{attribute 'linkalways'}
{attribute 'no_explicit_call' := 'This FB is a CLASS and must be accessed using methods or properties'}
{attribute 'enable_dynamic_creation'}
FUNCTION_BLOCK Node_F_VN_LocateCircularArcExp2 EXTENDS VisionNode
VAR
    ipSrcImage : _ITcVnImage;
    stCircularArc : _TcVnCircularArc;
    aCenter : _TcVnPoint2_REAL;
    fSearchRadius : _REAL(0.0);
    fArcDirectionRad : _LREAL(0.0);
    eEdgeDirection : _ETcVnEdgeDirection(ETcVnEdgeDirection.TCVN_ED_DARK_TO_LIGHT);
    fMinStrength : _REAL(0.0);
    fAngleStepRad : _LREAL(0.1);
    nMaxThickness : _UDINT(10);
    bInvertSearchDirection : _BOOL(FALSE);
    nSubpixelsIterations : _UDINT(10);
    fApproxPrecision : _REAL(0.001);
    eAlgorithm : _ETcVnEdgeDetectionAlgorithm(ETcVnEdgeDetectionAlgorithm.TCVN_EDA_INTERPOLATION);
    ipContourPoints : _ITcVnContainer;
    fRangeCutoffFactor : _REAL(0.135);
    hrPrev : _HRESULT(S_OK);
    hresult : _HRESULT(S_OK);
END_VAR

METHOD PUBLIC Clone : I_Node
VAR
    pNode : POINTER TO Node_F_VN_LocateCircularArcExp2;
END_VAR
pNode := __NEW(Node_F_VN_LocateCircularArcExp2);
Clone := pNode^;
END_METHOD

METHOD FB_init : BOOL
VAR_INPUT
    bInitRetains : BOOL;
    bInCopyCode : BOOL;
END_VAR
AddInput('ipSrcImage', ipSrcImage);
AddOutput('stCircularArc', stCircularArc);
AddInput('aCenter', aCenter);
AddParameter('fSearchRadius', fSearchRadius);
AddParameter('fArcDirectionRad', fArcDirectionRad);
AddParameter('eEdgeDirection', eEdgeDirection);
AddParameter('fMinStrength', fMinStrength);
AddParameter('fAngleStepRad', fAngleStepRad);
AddParameter('nMaxThickness', nMaxThickness);
AddParameter('bInvertSearchDirection', bInvertSearchDirection);
AddParameter('nSubpixelsIterations', nSubpixelsIterations);
AddParameter('fApproxPrecision', fApproxPrecision);
AddParameter('eAlgorithm', eAlgorithm);
AddOutput('ipContourPoints', ipContourPoints);
AddParameter('fRangeCutoffFactor', fRangeCutoffFactor);
AddInput('hrPrev', hrPrev);
AddOutput('aCenter', aCenter);
AddOutput('hresult', hresult);
END_METHOD

METHOD PROTECTED OnExecute
hresult.Value := F_VN_LocateCircularArcExp2(
    ipSrcImage := ipSrcImage.Value,
    stCircularArc := stCircularArc.Value,
    aCenter := aCenter.Value,
    fSearchRadius := fSearchRadius.Value,
    fArcDirectionRad := fArcDirectionRad.Value,
    eEdgeDirection := eEdgeDirection.Value,
    fMinStrength := fMinStrength.Value,
    fAngleStepRad := fAngleStepRad.Value,
    nMaxThickness := nMaxThickness.Value,
    bInvertSearchDirection := bInvertSearchDirection.Value,
    nSubpixelsIterations := nSubpixelsIterations.Value,
    fApproxPrecision := fApproxPrecision.Value,
    eAlgorithm := eAlgorithm.Value,
    ipContourPoints := ipContourPoints.Value,
    fRangeCutoffFactor := fRangeCutoffFactor.Value,
    hrPrev := hrPrev.Value);
END_METHOD

METHOD PUBLIC PreExecutionCheck
VAR_INPUT
    Check : I_PreExecutionChecks;
END_VAR
VAR
    width : UDINT;
    height : UDINT;
    cx : REAL;
    cy : REAL;
END_VAR
Check.IsTrue(ipSrcImage.IsValid, 'ipSrcImage must contain an image');
Check.IsTrue(ipSrcImage.HasChannelCount(1), 'ipSrcImage must contain 1 channel');

// Input search radius (starting FROM aCenter, should be greater than the actual radius but
// aCenter + fSearchRadius should be within the image borders)
ipSrcImage.TryGetWidth(width);
ipSrcImage.TryGetHeight(height);

Check.IsTrue((width > 0), 'ipSrcImage have valid width');
Check.IsTrue((height > 0), 'ipSrcImage have valid height');
Check.IsTrue(fSearchRadius.Value > 0, 'fSearchRadius must be > 0');

cx := aCenter.Value[0];
cy := aCenter.Value[1];

Check.IsTrue(cx - fSearchRadius.Value >= 0, 'Search radius exceeds left border');
Check.IsTrue(cy - fSearchRadius.Value >= 0, 'Search radius exceeds top border');
Check.IsTrue(cx + fSearchRadius.Value < UDINT_TO_REAL(width), 'Search radius exceeds right border');
Check.IsTrue(cy + fSearchRadius.Value < UDINT_TO_REAL(height), 'Search radius exceeds bottom border');

// Input search starting direction in radian. Valid range is [-pi, +pi], where right is 0 rad,
// top is -pi/2 rad and bottom +pi/2 rad. The circular arc should at least be valid in range
// fArcDirectionRad +- 4 * fAngleStepRad.
Check.IsTrue(fAngleStepRad.Value > 0.0, 'fAngleStepRad must be greater than 0');
Check.IsTrue(fArcDirectionRad.Value >= -PI AND fArcDirectionRad.Value <= PI, 'fArcDirectionRad must be in [-pi, +pi]');
Check.IsTrue(fArcDirectionRad.Value - 4.0 * fAngleStepRad.Value >= -PI, 'fArcDirectionRad - 4 * fAngleStepRad must be >= -pi');
Check.IsTrue(fArcDirectionRad.Value + 4.0 * fAngleStepRad.Value <=  PI, 'fArcDirectionRad + 4 * fAngleStepRad must be <= +pi');

Check.IsTrue(nMaxThickness.Value > 0, 'nMaxThickness must be at least 1');
Check.IsTrue(nSubpixelsIterations.Value > 0, 'nSubpixelsIterations must be greater than 0');
Check.IsTrue((eAlgorithm.Value = ETcVnEdgeDetectionAlgorithm.TCVN_EDA_INTERPOLATION) OR
             (fApproxPrecision.Value > 0.0), 'fApproxPrecision must be greater than 0 for the approximation algorithms');
END_METHOD

END_FUNCTION_BLOCK

(* stored: Version 1.1.0.1, ProductVersion 3.1.4026.19
   POU Node_F_VN_LocateCircularArcExp2: Id {1be000da-add6-43f0-9ba6-a87486481eec}, SpecialFunc None
   Folder Constructor: Id {807676ad-8b0d-4925-b74e-737a0f55abb3}
   Method Clone: Id {9310f832-a3d3-4cdf-bc11-eeb6dfa89e95}
   Method FB_init: Id {19bc087f-2c99-421c-bfb9-ce260d592277}
   Method OnExecute: Id {c4d1ac29-1bfe-4f5a-af4c-69bcad40524c}
   Method PreExecutionCheck: Id {02b13a84-0465-4fe1-a224-6e8cd5842833} *)
